// TIA Portal V16 program export: 1 tag tables, 0 data types, 16 data blocks, 4 code blocks (in call order from the OBs), 0 instance data blocks

VAR_GLOBAL   // PLC tag table "Default tag table"
END_VAR

DATA_BLOCK "BlockIncrementer_DB"
{ S7_Optimized_Access := 'TRUE' }
VERSION : 0.1
NON_RETAIN
"BlockIncrementer"

BEGIN

END_DATA_BLOCK

DATA_BLOCK "Main_Safety_RTG1_DB"
{ S7_Optimized_Access := 'TRUE' }
NAME : FUSI
VERSION : 0.1
NON_RETAIN
"Main_Safety_RTG1"

BEGIN

END_DATA_BLOCK

DATA_BLOCK "MyCounter_DB0"
{ S7_Optimized_Access := 'TRUE' }
VERSION : 0.1
NON_RETAIN
"MyCounter"

BEGIN

END_DATA_BLOCK

DATA_BLOCK "MyCounter_DB1"
{ S7_Optimized_Access := 'TRUE' }
VERSION : 0.1
NON_RETAIN
"MyCounter"

BEGIN

END_DATA_BLOCK

DATA_BLOCK "F_SystemInfo_DB"
{ S7_Optimized_Access := 'TRUE' }
NAME : F_GLOBDB
VERSION : 0.1
NON_RETAIN
   VAR 
      FCCValue : DWord;
   END_VAR


BEGIN

END_DATA_BLOCK

DATA_BLOCK "RTG1SysInfo"
{InstructionName := 'F_CTRL1';
 LibVersion := '2.2';
 S7_Optimized_Access := 'TRUE' }
AUTHOR : SafeSys
FAMILY : F_CTRL
NAME : F_CTRL_1
VERSION : 2.2
NON_RETAIN
F_CTRL1

BEGIN
   F_SYSINFO.F_PROG_SIG := DW#16#832DEE38;
   F_SYSINFO.F_PROG_DAT := DTL#2021-8-4-22:50:56.862582800;
   F_SYSINFO.F_RTG_SIG := DW#16#F5BD20EF;
   F_SYSINFO.F_RTG_DAT := DTL#2021-8-4-22:50:56.862582800;
   F_SYSINFO.VERS_S7SAF := DW#16#16000000;
   dnMODE_C := 19127;
   dnDB_INIT_C := 70557;
   dnMOD_MODE_C := 34321;
   dnPLCSIM_MODE_C := 20664;
   dnACT_MOD_MODE_C := 27190;
   lnDIFF_C := 35673;
   lnDIFF_MTIME_C := 22975;
   nMAX_CYC := 120;
   dnMAX_CYC_C := 3819182;
   nWARN_CYC := 110;
   dwFCC_VALUE := DW#16#B0695B45;
   dnS_TIM_C := 14080;
   dnS_TIM_ALT_C := 33803;
   dnS_TIM100_CACHE_C := 32709;
   dnS_TIM100_USE_C := 25382;
   dnS_TIM1000_CACHE_C := 26562;
   dnS_TIM1000_USE_C := 41245;
   dnS_DIFF_C := 14080;
   dnS_DIFF100_C := 14080;
   dnS_DIFF1000_C := 14080;
   lnF_TIM_SFC_C := 14080;
   lnF_TIM_SFC_ALT_C := 27889;
   dnF_TIM_C := 14080;
   dnF_TIM_ALT_C := 23998;
   dnF_TIM100_CACHE_C := 26848;
   dnF_TIM100_USE_C := 25044;
   dnF_TIM1000_CACHE_C := 25507;
   dnF_TIM1000_USE_C := 23558;
   dnF_DIFF_C := 14080;
   dnF_DIFF100_C := 14080;
   dnF_DIFF1000_C := 14080;
   dnCONTROL_TIM100_C := 39214;
   dnCONTROL_TIM1000_C := 24463;
   dnTOL_C := 14080;
   dwF_PROG_SIG_DAT_SIG := DW#16#B04411D9;
   dwF_RTG_SIG_DAT_SIG := DW#16#C6D4DF0E;
   wRTG_NO := W#16#1;

END_DATA_BLOCK

DATA_BLOCK "DB1_C"
{ S7_Optimized_Access := 'TRUE' }
NAME : FCDI
VERSION : 0.1
NON_RETAIN
"FB1_C"

BEGIN
   dnCALLCHECK_C := 61159;
   dnTRACER_START := 20389;
   dnGCTX_DBNUMBER := 30010;

END_DATA_BLOCK

DATA_BLOCK "DB3_C"
{ S7_Optimized_Access := 'TRUE' }
NAME : FCDI
VERSION : 0.1
NON_RETAIN
"FB2_C"

BEGIN
   increment_C := 111444;
   counter_C := 92146;
   dnCALLCHECK_C := 87957;
   dnTRACER_START := 20944;
   dnGCTX_DBNUMBER := 30011;

END_DATA_BLOCK

DATA_BLOCK "DB4_C"
{ S7_Optimized_Access := 'TRUE' }
NAME : FCDI
VERSION : 0.1
NON_RETAIN
"FB2_C"

BEGIN
   increment_C := 138146;
   counter_C := 118848;
   dnCALLCHECK_C := 114659;
   dnTRACER_START := 20944;
   dnGCTX_DBNUMBER := 30011;

END_DATA_BLOCK

DATA_BLOCK "FB1_C_GCTX_DB"
{ S7_Optimized_Access := 'TRUE' }
NAME : F_GLOBDB
VERSION : 0.1
NON_RETAIN
   VAR 
      GCTX_DINT { ExternalAccessible := 'False'; ExternalVisible := 'False'; ExternalWritable := 'False'} : Array[0..0, 0..4] of DInt;
   END_VAR


BEGIN
   GCTX_DINT[0,0] := 1885684513;
   GCTX_DINT[0,1] := 32;
   GCTX_DINT[0,2] := 13215;
   GCTX_DINT[0,3] := 64;
   GCTX_DINT[0,4] := 96;

END_DATA_BLOCK

DATA_BLOCK "FB2_C_GCTX_DB"
{ S7_Optimized_Access := 'TRUE' }
NAME : F_GLOBDB
VERSION : 0.1
NON_RETAIN
   VAR 
      GCTX_DINT { ExternalAccessible := 'False'; ExternalVisible := 'False'; ExternalWritable := 'False'} : Array[0..2, 0..0] of DInt;
   END_VAR


BEGIN
   GCTX_DINT[0,0] := 1885664965;
   GCTX_DINT[1,0] := 19548;
   GCTX_DINT[2,0] := 1885684513;

END_DATA_BLOCK

DATA_BLOCK "FB32770_IDB_C"
{InstructionName := 'F_CTRLD';
 LibVersion := '1.4';
 S7_Optimized_Access := 'TRUE' }
AUTHOR : SafeSys
FAMILY : F_CTRL
NAME : F_CTRL_D
VERSION : 1.2
NON_RETAIN
F_CTRLD

BEGIN

END_DATA_BLOCK

DATA_BLOCK "FB32771_IDB_C"
{InstructionName := 'F_CTRL2';
 LibVersion := '1.4';
 S7_Optimized_Access := 'TRUE' }
AUTHOR : SafeSys
FAMILY : F_CTRL
NAME : F_CTRL_2
VERSION : 1.2
NON_RETAIN
F_CTRL2

BEGIN
   dnMOD_MODE_C := 55467;
   dnP_FOB := 8966;
   wRTG_NO := W#16#1;

END_DATA_BLOCK

DATA_BLOCK "FB32772_IDB_C"
{InstructionName := 'F_ETLI';
 LibVersion := '2.0';
 S7_Optimized_Access := 'TRUE' }
AUTHOR : SafeSys
FAMILY : F_CTRL
NAME : F_ET_LI
VERSION : 2.0
NON_RETAIN
F_ETLI

BEGIN

END_DATA_BLOCK

DATA_BLOCK "FB32773_IDB_C"
{InstructionName := 'F_CTRLRT';
 LibVersion := '1.3';
 S7_Optimized_Access := 'TRUE' }
AUTHOR : SafeSys
FAMILY : F_CTRL
NAME : F_CTRLRT
VERSION : 1.0
NON_RETAIN
F_CTRLRT

BEGIN

END_DATA_BLOCK

DATA_BLOCK "FOB_RTG1_GCTX_DB"
{ S7_Optimized_Access := 'TRUE' }
NAME : F_GLOBDB
VERSION : 0.1
NON_RETAIN
   VAR 
      GCTX_DINT { ExternalAccessible := 'False'; ExternalVisible := 'False'; ExternalWritable := 'False'} : Array[0..0, 0..2] of DInt;
   END_VAR


BEGIN
   GCTX_DINT[0,0] := 1885670433;
   GCTX_DINT[0,1] := 32;
   GCTX_DINT[0,2] := 8609;

END_DATA_BLOCK

ORGANIZATION_BLOCK "Main"   // OB1, LAD, ProgramCycle
TITLE = "Main Program Sweep (Cycle)"
{ S7_Optimized_Access := 'TRUE' }
VERSION : 0.1
// stored: AutoNumber true, IsIECCheckEnabled false, SetENOAutomatically false
   VAR_INPUT
      Initial_Call : Bool;   // Initial call of this OB
      Remanence : Bool;   // =True, if remanent data are available
   END_VAR
BEGIN
END_ORGANIZATION_BLOCK

FUNCTION_BLOCK "BlockIncrementer"   // FB3, F_FBD
{ S7_Optimized_Access := 'TRUE' }
VERSION : 0.1
// stored: AutoNumber true, IsIECCheckEnabled false, UDAEnableTagReadback false
   VAR
      "a" : "MyCounter";
      "b" : "MyCounter";
   END_VAR
BEGIN

REGION Network 1
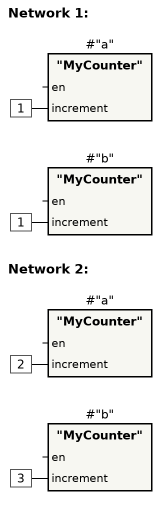
   #"a"(increment := 1);   // "MyCounter"
   #"b"(increment := 1);   // "MyCounter"
END_REGION

REGION Network 2
   #"a"(increment := 2);   // "MyCounter"
   #"b"(increment := 3);   // "MyCounter"
END_REGION
END_FUNCTION_BLOCK

FUNCTION_BLOCK "MyCounter"   // FB2, F_FBD
{ S7_Optimized_Access := 'TRUE' }
VERSION : 0.1
// stored: AutoNumber true, IsIECCheckEnabled false, UDAEnableTagReadback false
   VAR_INPUT
      increment : Int;
   END_VAR
   VAR
      "counter" : Int;
   END_VAR
BEGIN

REGION Network 1
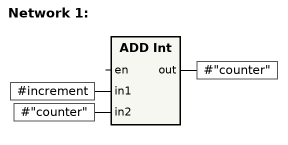
   #"counter" := #increment + #"counter";
END_REGION
END_FUNCTION_BLOCK

FUNCTION_BLOCK "Main_Safety_RTG1"   // FB1, F_FBD
{ S7_Optimized_Access := 'TRUE' }
VERSION : 0.1
// stored: AutoNumber false, IsIECCheckEnabled false, UDAEnableTagReadback false
BEGIN

REGION Network 1
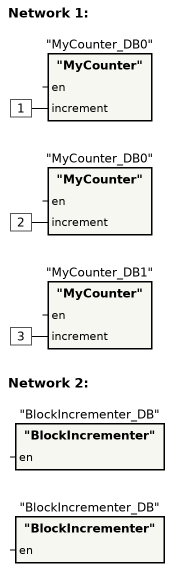
   "MyCounter_DB0"(increment := 1);   // "MyCounter"
   "MyCounter_DB0"(increment := 2);   // "MyCounter"
   "MyCounter_DB1"(increment := 3);   // "MyCounter"
END_REGION

REGION Network 2
   "BlockIncrementer_DB"();   // "BlockIncrementer"
   "BlockIncrementer_DB"();   // "BlockIncrementer"
END_REGION
END_FUNCTION_BLOCK
